(* IEC 61131-3 sources: RL_MAR/experiments/comparison/llm4plc/results/gpt-4o_20260507_114630/20260507_122022, 3 files *)

(* ---- generated_code_iteration_0.st ---- *)
START_ST
FUNCTION_BLOCK FruitJuicingBottling
VAR_INPUT
    StartButton : BOOL; (* Input for starting the process *)
    StopButton : BOOL; (* Input for stopping the process *)
    FruitSelected : BOOL; (* Input indicating fruit selection *)
END_VAR
VAR_OUTPUT
    JuiceProcessing : BOOL; (* Output for controlling juice extraction *)
    BottleFilling : BOOL; (* Output for controlling bottle filling *)
    CapPlacement : BOOL; (* Output for placing caps on bottles *)
    Packaging : BOOL; (* Output for packaging filled bottles *)
    ProcessInProgress : BOOL; (* Indicator for an ongoing process *)
END_VAR
VAR
    state : INT := 0; (* Current state of the system, initialized to STATE 0 (IDLE) *)
    prevState : INT := -1; (* Previous state of the system, initialized to an invalid state *)
END_VAR

(* State Definitions *)
CONST
    STATE_IDLE : INT := 0; (* System is idle *)
    STATE_PROCESS_RUNNING : INT := 1; (* System is running the process *)
    STATE_STOPPING : INT := 2; (* System is stopping *)
END_VAR

(* Main Logic *)
CASE state OF
    (* STATE 0: IDLE *)
    STATE_IDLE:
        (* Set outputs to FALSE *)
        JuiceProcessing := FALSE;
        BottleFilling := FALSE;
        CapPlacement := FALSE;
        Packaging := FALSE;
        ProcessInProgress := FALSE;

        (* Transition to STATE 1 if start conditions are met *)
        IF StartButton AND FruitSelected AND NOT ProcessInProgress THEN
            prevState := state; (* Store the current state as the previous state *)
            state := STATE_PROCESS_RUNNING; (* Transition to STATE 1 *)
        END_IF;

    (* STATE 1: PROCESS_RUNNING *)
    STATE_PROCESS_RUNNING:
        (* Set outputs to TRUE *)
        JuiceProcessing := TRUE;
        BottleFilling := TRUE;
        CapPlacement := TRUE;
        Packaging := TRUE;
        ProcessInProgress := TRUE;

        (* Transition to STATE 2 if stop conditions are met *)
        IF StopButton OR NOT FruitSelected THEN
            prevState := state; (* Store the current state as the previous state *)
            state := STATE_STOPPING; (* Transition to STATE 2 *)
        END_IF;

    (* STATE 2: STOPPING *)
    STATE_STOPPING:
        (* Set outputs to FALSE *)
        JuiceProcessing := FALSE;
        BottleFilling := FALSE;
        CapPlacement := FALSE;
        Packaging := FALSE;
        ProcessInProgress := FALSE;

        (* Transition back to STATE 0 once stopping is complete *)
        prevState := state; (* Store the current state as the previous state *)
        state := STATE_IDLE; (* Transition to STATE 0 *)

    ELSE
        (* Default case to handle unexpected states *)
        state := STATE_IDLE; (* Reset to STATE 0 *)
END_CASE;

END_FUNCTION_BLOCK
END_ST

(* ---- generated_code_iteration_1.st ---- *)
START_REASON
The feedback indicates that the `CONST` section used for defining state constants (`STATE_IDLE`, `STATE_PROCESS_RUNNING`, `STATE_STOPPING`) is not valid in CODESYS. Instead, constants should be defined within the `VAR`, `VAR_INPUT`, `VAR_OUTPUT`, or `VAR_IN_OUT` sections. To resolve this, the constants will be moved to the `VAR` section, as they are internal to the function block and do not require external input or output.

Additionally, I will ensure the code adheres to proper syntax and structure for CODESYS compliance while maintaining the functionality described in the original requirements.
END_REASON

START_ST
FUNCTION_BLOCK FruitJuicingBottling
VAR_INPUT
    StartButton : BOOL; (* Input for starting the process *)
    StopButton : BOOL; (* Input for stopping the process *)
    FruitSelected : BOOL; (* Input indicating fruit selection *)
END_VAR
VAR_OUTPUT
    JuiceProcessing : BOOL; (* Output for controlling juice extraction *)
    BottleFilling : BOOL; (* Output for controlling bottle filling *)
    CapPlacement : BOOL; (* Output for placing caps on bottles *)
    Packaging : BOOL; (* Output for packaging filled bottles *)
    ProcessInProgress : BOOL; (* Indicator for an ongoing process *)
END_VAR
VAR
    state : INT := 0; (* Current state of the system, initialized to STATE 0 (IDLE) *)
    prevState : INT := -1; (* Previous state of the system, initialized to an invalid state *)

    (* State Definitions *)
    STATE_IDLE : INT := 0; (* System is idle *)
    STATE_PROCESS_RUNNING : INT := 1; (* System is running the process *)
    STATE_STOPPING : INT := 2; (* System is stopping *)
END_VAR

(* Main Logic *)
CASE state OF
    (* STATE 0: IDLE *)
    STATE_IDLE:
        (* Set outputs to FALSE *)
        JuiceProcessing := FALSE;
        BottleFilling := FALSE;
        CapPlacement := FALSE;
        Packaging := FALSE;
        ProcessInProgress := FALSE;

        (* Transition to STATE 1 if start conditions are met *)
        IF StartButton AND FruitSelected AND NOT ProcessInProgress THEN
            prevState := state; (* Store the current state as the previous state *)
            state := STATE_PROCESS_RUNNING; (* Transition to STATE 1 *)
        END_IF;

    (* STATE 1: PROCESS_RUNNING *)
    STATE_PROCESS_RUNNING:
        (* Set outputs to TRUE *)
        JuiceProcessing := TRUE;
        BottleFilling := TRUE;
        CapPlacement := TRUE;
        Packaging := TRUE;
        ProcessInProgress := TRUE;

        (* Transition to STATE 2 if stop conditions are met *)
        IF StopButton OR NOT FruitSelected THEN
            prevState := state; (* Store the current state as the previous state *)
            state := STATE_STOPPING; (* Transition to STATE 2 *)
        END_IF;

    (* STATE 2: STOPPING *)
    STATE_STOPPING:
        (* Set outputs to FALSE *)
        JuiceProcessing := FALSE;
        BottleFilling := FALSE;
        CapPlacement := FALSE;
        Packaging := FALSE;
        ProcessInProgress := FALSE;

        (* Transition back to STATE 0 once stopping is complete *)
        prevState := state; (* Store the current state as the previous state *)
        state := STATE_IDLE; (* Transition to STATE 0 *)

    ELSE
        (* Default case to handle unexpected states *)
        state := STATE_IDLE; (* Reset to STATE 0 *)
END_CASE;

END_FUNCTION_BLOCK
END_ST

(* ---- generated_code_iteration_2.st ---- *)
START_REASON
The feedback indicates that the `CASE` statement in the code failed CODESYS compiler validation due to an issue with the labels used in the `CASE` statement. Specifically, the labels in the `CASE` statement must be integer constants or literal values, but the current implementation uses symbolic constants (`STATE_IDLE`, `STATE_PROCESS_RUNNING`, `STATE_STOPPING`) defined in the `VAR` section.

To resolve this issue, the symbolic constants will be replaced with literal integer values directly within the `CASE` statement. This ensures compliance with CODESYS syntax requirements while maintaining the intended functionality of the state machine.

Additionally, I will verify that all other aspects of the code adhere to proper syntax and structure for CODESYS compliance.
END_REASON

START_ST
FUNCTION_BLOCK FruitJuicingBottling
VAR_INPUT
    StartButton : BOOL; (* Input for starting the process *)
    StopButton : BOOL; (* Input for stopping the process *)
    FruitSelected : BOOL; (* Input indicating fruit selection *)
END_VAR
VAR_OUTPUT
    JuiceProcessing : BOOL; (* Output for controlling juice extraction *)
    BottleFilling : BOOL; (* Output for controlling bottle filling *)
    CapPlacement : BOOL; (* Output for placing caps on bottles *)
    Packaging : BOOL; (* Output for packaging filled bottles *)
    ProcessInProgress : BOOL; (* Indicator for an ongoing process *)
END_VAR
VAR
    state : INT := 0; (* Current state of the system, initialized to STATE 0 (IDLE) *)
    prevState : INT := -1; (* Previous state of the system, initialized to an invalid state *)
END_VAR

(* Main Logic *)
CASE state OF
    (* STATE 0: IDLE *)
    0:
        (* Set outputs to FALSE *)
        JuiceProcessing := FALSE;
        BottleFilling := FALSE;
        CapPlacement := FALSE;
        Packaging := FALSE;
        ProcessInProgress := FALSE;

        (* Transition to STATE 1 if start conditions are met *)
        IF StartButton AND FruitSelected AND NOT ProcessInProgress THEN
            prevState := state; (* Store the current state as the previous state *)
            state := 1; (* Transition to STATE 1 *)
        END_IF;

    (* STATE 1: PROCESS_RUNNING *)
    1:
        (* Set outputs to TRUE *)
        JuiceProcessing := TRUE;
        BottleFilling := TRUE;
        CapPlacement := TRUE;
        Packaging := TRUE;
        ProcessInProgress := TRUE;

        (* Transition to STATE 2 if stop conditions are met *)
        IF StopButton OR NOT FruitSelected THEN
            prevState := state; (* Store the current state as the previous state *)
            state := 2; (* Transition to STATE 2 *)
        END_IF;

    (* STATE 2: STOPPING *)
    2:
        (* Set outputs to FALSE *)
        JuiceProcessing := FALSE;
        BottleFilling := FALSE;
        CapPlacement := FALSE;
        Packaging := FALSE;
        ProcessInProgress := FALSE;

        (* Transition back to STATE 0 once stopping is complete *)
        prevState := state; (* Store the current state as the previous state *)
        state := 0; (* Transition to STATE 0 *)

    ELSE
        (* Default case to handle unexpected states *)
        state := 0; (* Reset to STATE 0 *)
END_CASE;

END_FUNCTION_BLOCK
END_ST
